// TIA Portal V16 export
// export: Created 2023-03-29T11:03:46.0312675Z, ExportSetting WithDefaults, DisplayName Totally Integrated Automation Portal, DisplayVersion V16 Update 6, DisplayName TIA Portal Version Control Interface, DisplayVersion V16 Update 2, DisplayName TIA Portal Openness, DisplayVersion V16 Update 6, DisplayName STEP 7 Professional, DisplayVersion V16 Update 6, DisplayName STEP 7 Safety, DisplayVersion V16, DisplayName WinCC Advanced, DisplayVersion V16 Update 6
VAR_GLOBAL   // PLC tag table "Zasuwy"
   isAutPumping AT %M80.6 : Bool;   // wybrana opcja automatycznego sterowania pompowanie lub dosilanie
   isPumping AT %M80.4 : Bool;   // wybrana opcja przepompowywanie na miasto
   isTime_FillingOn AT %M90.4 : Bool;   // znacznik start napełnianie
   isTime_FillingOff AT %M90.5 : Bool;   // znacznik stop napełnianie
   isTime_EptyingOn AT %M90.6 : Bool;   // znacznik start przetłaczanie
   isRecharging AT %M80.5 : Bool;   // wybrana opcja dosilania na magistralę
   isTime_EptyingOff AT %M90.7 : Bool;   // znacznik stop przetłaczanie
   inputREM_Zasuwy AT %M50.4 : Bool;   // znacznik wejście zdalane
   isManual AT %M81.1 : Bool;   // tryb sterowania manualny
   memTriggerClose_setValue_Z11 AT %M90.1 : Bool;   // pamięć zbocza przekazania nowego meldunku dla otwierania
   memTriggerOpen_setValue_Z10 AT %M90.0 : Bool;   // pamięć zbocza przekazania nowego meldunku
END_VAR
